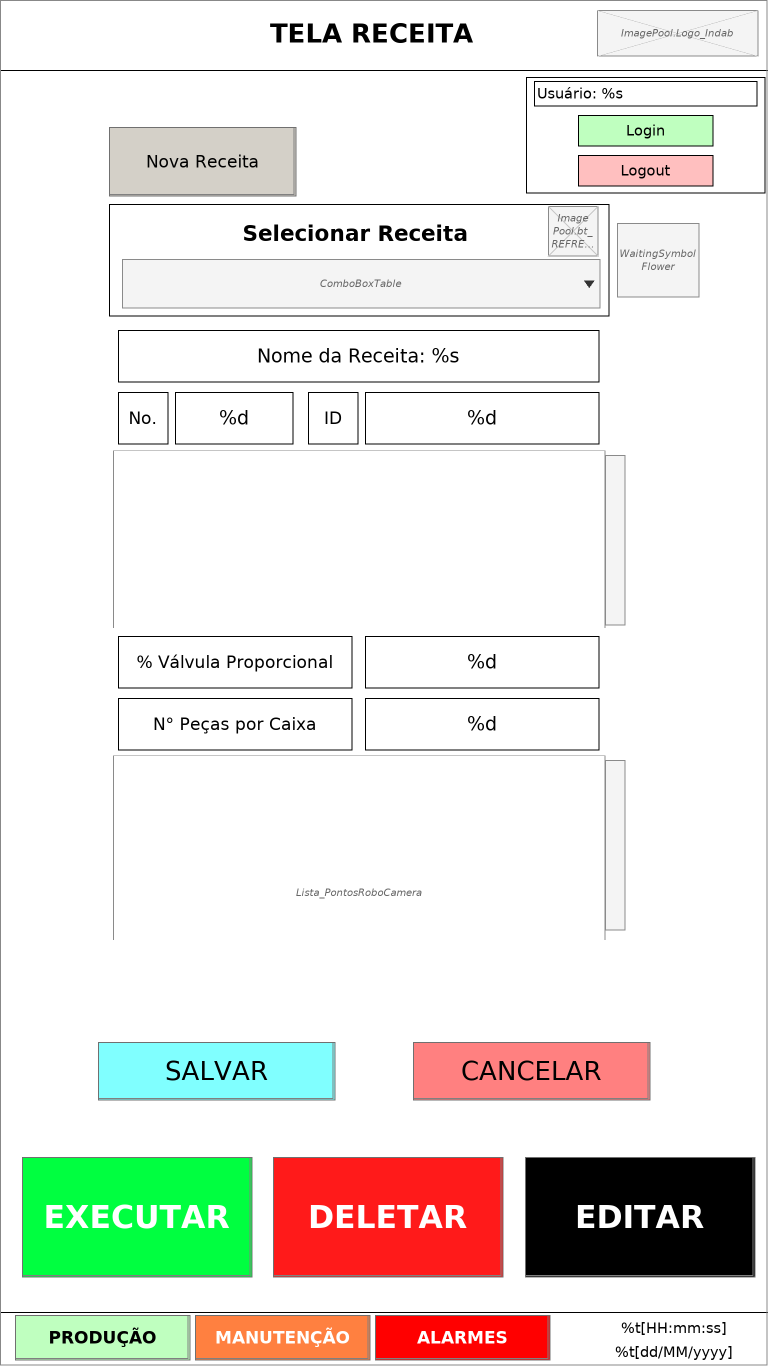
VISUALIZATION Tela_Receita  // 768x1366, background image __VisualizationStyle.CheckboxChecked
    Frame (113,450 492x675)
        shows Lista_PontosSolda()
        shows Lista_PontosRoboCamera()
        p2738717112: Main_Receita.ScrollScreen_PontosSolda
    Rectangle (-1,628 768x500)
    Rectangle (-1,628 768x737)
    Frame (113,755 492x275)
        shows Lista_PontosRoboCamera()
        shows Lista_PontosRoboCamera()
        p2738717112: Main_Receita.ScrollScreen_PontosSolda
    Rectangle (-1,0 768x450)
    Rectangle (109,204 500x112)
    Line (0,70) (768,70)
    Image (597,10 161x46), image: ImagePool.Logo_Indab
    Label (153,7 437x53), "TELA RECEITA"
    ComboBoxTable (122,259 478x49), variable: Recipe_select_int, input disabled if: b_editar_receita or b_criar_receita, data array: Recipe_names_saved
        p1128707560: Main_Receita.Item_livre
        p3854506369: Recipe_names_saved[INDEX]
    Rectangle (118,330 481x52), "Nome da Receita: %s", text variable: Recipe_name_Select, input disabled if: Not b_editar_receita and Not b_criar_receita
        OnMouseClick: write the text variable via Default
    Rectangle (526,77 239x116)
    Rectangle (578,115 135x31), "Login"
        OnMouseClick: VisuUserMgmt Type=Login
    Rectangle (578,155 135x31), "Logout"
        OnMouseClick: VisuUserMgmt Type=Logout
    Rectangle (534,81 223x25), "Usuário: %s", text variable: UserName
    Button (109,127 187x69), "Nova Receita"
        OnMouseClick: execute { b_criar_receita := TRUE; }
    Label (137,207 437x53), "Selecionar Receita"
    WaitingSymbolFlower (617,223 82x74), invisible if: Not Simbolo_Atualizacao
    Image (548,206 50x50), image: ImagePool.bt_REFRESH
        OnMouseClick: execute { bRead := TRUE; }
    Scrollbar (605,455 20x170), invisible if: Recipe_Pontos_Solda_Select<=3
        p2245068023: Main_Receita.LengthScrollBar_PontosSolda
        p1057716461: Main_Receita.ScrollBar_PontosSolda
    Rectangle (365,392 234x52), "%d", text variable: Recipe_ID_Select, input disabled if: Not b_editar_receita and Not b_criar_receita
        OnMouseClick: write the text variable via Default
    Rectangle (118,392 50x52), "No."
    Rectangle (175,392 118x52), "%d", text variable: Recipe_No_Select, input disabled if: Not b_editar_receita and Not b_criar_receita
        OnMouseClick: write the text variable via Default
    Rectangle (308,392 50x52), "ID"
    Scrollbar (605,760 20x170), invisible if: Recipe_Pontos_Camera_Select<=3
        p2245068023: Main_Receita.LengthScrollBar_PontosCamera
        p1057716461: Main_Receita.ScrollBar_PontosCamera
    Rectangle (-1,630 768x125)
    Rectangle (118,636 234x52), "% Válvula Proporcional"
    Rectangle (365,636 234x52), "%d", text variable: Recipe_Valvula_Proporcional_Select, input disabled if: Not b_editar_receita and Not b_criar_receita
        OnMouseClick: write the text variable via Default
    Rectangle (365,698 234x52), "%d", text variable: Recipe_Pecas_Caixa_Select, input disabled if: Not b_editar_receita and Not b_criar_receita
        OnMouseClick: write the text variable via Default
    Rectangle (118,698 234x52), "N° Peças por Caixa"
    Line (0,1312) (768,1312)
    Rectangle (584,1340 180x24), "%t[dd/MM/yyyy]"
    Rectangle (584,1316 180x24), "%t[HH:mm:ss]"
    Rectangle (-1,940 768x365)
    Button (525,1157 230x120), "EDITAR", input disabled if: b_criar_receita
        OnMouseClick: execute { b_editar_receita := TRUE; }
    Button (22,1157 230x120), "EXECUTAR", input disabled if: b_editar_receita
        OnMouseClick: execute { b_executar_receita := TRUE; }
    Button (273,1157 230x120), "DELETAR", input disabled if: Not b_editar_receita
        OnMouseClick: execute { b_deletar_receita := TRUE; }
    Button (98,1042 237x58), "SALVAR", invisible if: Not b_editar_receita AND Not b_criar_receita
        OnMouseClick: execute { b_salvar_receita := TRUE; }
    Button (413,1042 237x58), "CANCELAR", invisible if: Not b_editar_receita AND NOT b_criar_receita
        OnMouseClick: execute { b_cancelar_receita := TRUE; }
    Button (15,1315 175x45), "PRODUÇÃO"
        OnMouseClick: change screen: Tela_Producao
    Button (195,1315 175x45), "MANUTENÇÃO"
        OnMouseClick: change screen: Tela_Manutencao
    Button (375,1315 175x45), "ALARMES"
        OnMouseClick: change screen: Tela_Alarmes_1
END_VISUALIZATION

(* stored: Version 1.1.0.1, ProductVersion 3.1.4024.11
   Visu Tela_Receita: Id {2db49080-364d-4b18-a310-0c063c4faa6f} *)
